ABB RAPID module: 8947b821.mod

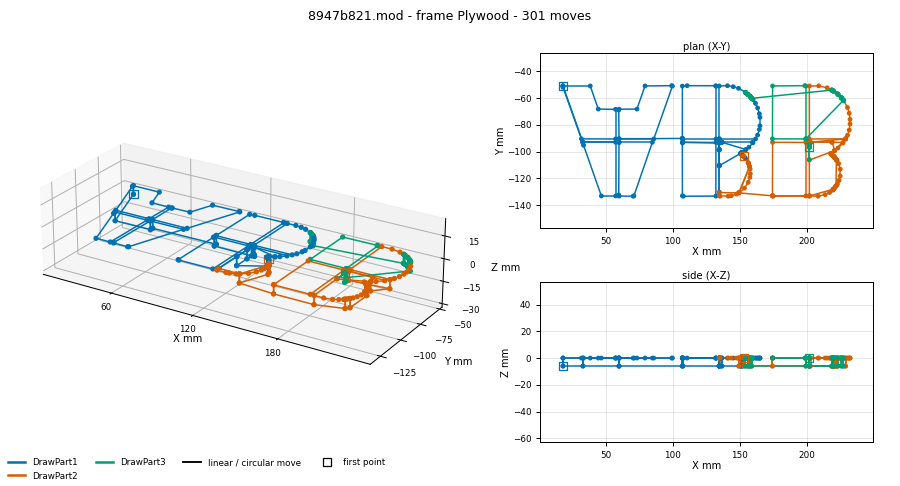
[picture p0: tool path of 8947b821.mod in frame Plywood, 301 of 303 moves have a stored position in this frame; points joined in program order, loops and branches not executed]
MODULE ImageDraw
  ! Generated 2026-10-07 09:33 for ABB GoFa CRB 15000-5/0.95: 40 strokes
  ! Page 250 x 180 mm. Work object Plywood: Z points DOWN, so pen-up is -Z and the tool uses orientation [1,0,0,0].
  ! Uses the tool 'tcp' and work object 'Plywood' that already exist on the controller.
  CONST robtarget pOrigin:=[[0,0,0],[1,0,0,0],[0,0,0,0],[9E9,9E9,9E9,9E9,9E9,9E9]];
  CONST jointtarget jHome:=[[0,0,0,0,30,0],[9E9,9E9,9E9,9E9,9E9,9E9]];
  CONST speeddata vTravel:=[250,200,5000,1000];

  PROC main()
    SingArea\Wrist;
    ConfL\Off;
    ConfJ\Off;
    MoveAbsJ jHome\NoEOffs,vTravel,fine,tcp;
    DrawPart1;
    DrawPart2;
    DrawPart3;
    MoveAbsJ jHome\NoEOffs,vTravel,fine,tcp;
  ENDPROC

  PROC DrawPart1()
    MoveL Offs(pOrigin,17.75,-50.83,-6.00),vTravel,z5,tcp\WObj:=Plywood;
    MoveL Offs(pOrigin,17.75,-50.83,-0.00),v60,z0,tcp\WObj:=Plywood;
    MoveL Offs(pOrigin,38.15,-50.83,-0.00),v40,z0,tcp\WObj:=Plywood;
    MoveL Offs(pOrigin,44.15,-68.12,-0.00),v40,z0,tcp\WObj:=Plywood;
    MoveL Offs(pOrigin,57.05,-68.32,-0.00),v40,z0,tcp\WObj:=Plywood;
    MoveL Offs(pOrigin,57.05,-90.47,-0.00),v40,z0,tcp\WObj:=Plywood;
    MoveL Offs(pOrigin,31.55,-90.38,-0.00),v40,z0,tcp\WObj:=Plywood;
    MoveL Offs(pOrigin,17.80,-51.83,-0.00),v40,z0,tcp\WObj:=Plywood;
    MoveL Offs(pOrigin,17.75,-50.83,-0.00),v40,fine,tcp\WObj:=Plywood;
    MoveL Offs(pOrigin,17.75,-50.83,-6.00),v60,z5,tcp\WObj:=Plywood;
    MoveL Offs(pOrigin,32.65,-92.97,-6.00),vTravel,z5,tcp\WObj:=Plywood;
    MoveL Offs(pOrigin,32.65,-92.97,-0.00),v60,z0,tcp\WObj:=Plywood;
    MoveL Offs(pOrigin,33.15,-95.18,-0.00),v40,z0,tcp\WObj:=Plywood;
    MoveL Offs(pOrigin,46.45,-133.07,-0.00),v40,z0,tcp\WObj:=Plywood;
    MoveL Offs(pOrigin,57.15,-133.07,-0.00),v40,z0,tcp\WObj:=Plywood;
    MoveL Offs(pOrigin,57.15,-92.97,-0.00),v40,z0,tcp\WObj:=Plywood;
    MoveL Offs(pOrigin,32.65,-92.97,-0.00),v40,fine,tcp\WObj:=Plywood;
    MoveL Offs(pOrigin,32.65,-92.97,-6.00),v60,z5,tcp\WObj:=Plywood;
    MoveL Offs(pOrigin,59.65,-92.97,-6.00),vTravel,z5,tcp\WObj:=Plywood;
    MoveL Offs(pOrigin,59.65,-92.97,-0.00),v60,z0,tcp\WObj:=Plywood;
    MoveL Offs(pOrigin,59.45,-132.38,-0.00),v40,z0,tcp\WObj:=Plywood;
    MoveL Offs(pOrigin,59.75,-133.18,-0.00),v40,z0,tcp\WObj:=Plywood;
    MoveL Offs(pOrigin,70.25,-133.27,-0.00),v40,z0,tcp\WObj:=Plywood;
    MoveL Offs(pOrigin,70.80,-132.98,-0.00),v40,z0,tcp\WObj:=Plywood;
    MoveL Offs(pOrigin,84.60,-92.97,-0.00),v40,z0,tcp\WObj:=Plywood;
    MoveL Offs(pOrigin,59.65,-92.97,-0.00),v40,fine,tcp\WObj:=Plywood;
    MoveL Offs(pOrigin,59.65,-92.97,-6.00),v60,z5,tcp\WObj:=Plywood;
    MoveL Offs(pOrigin,59.65,-90.38,-6.00),vTravel,z5,tcp\WObj:=Plywood;
    MoveL Offs(pOrigin,59.65,-90.38,-0.00),v60,z0,tcp\WObj:=Plywood;
    MoveL Offs(pOrigin,59.45,-68.78,-0.00),v40,z0,tcp\WObj:=Plywood;
    MoveL Offs(pOrigin,59.75,-68.22,-0.00),v40,z0,tcp\WObj:=Plywood;
    MoveL Offs(pOrigin,73.05,-68.12,-0.00),v40,z0,tcp\WObj:=Plywood;
    MoveL Offs(pOrigin,79.10,-50.83,-0.00),v40,z0,tcp\WObj:=Plywood;
    MoveL Offs(pOrigin,99.05,-50.62,-0.00),v40,z0,tcp\WObj:=Plywood;
    MoveL Offs(pOrigin,99.60,-50.92,-0.00),v40,z0,tcp\WObj:=Plywood;
    MoveL Offs(pOrigin,85.65,-90.47,-0.00),v40,z0,tcp\WObj:=Plywood;
    MoveL Offs(pOrigin,59.65,-90.38,-0.00),v40,fine,tcp\WObj:=Plywood;
    MoveL Offs(pOrigin,59.65,-90.38,-6.00),v60,z5,tcp\WObj:=Plywood;
    MoveL Offs(pOrigin,107.00,-90.07,-6.00),vTravel,z5,tcp\WObj:=Plywood;
    MoveL Offs(pOrigin,107.00,-90.07,-0.00),v60,z0,tcp\WObj:=Plywood;
    MoveL Offs(pOrigin,107.05,-50.92,-0.00),v40,z0,tcp\WObj:=Plywood;
    MoveL Offs(pOrigin,110.60,-50.62,-0.00),v40,z0,tcp\WObj:=Plywood;
    MoveL Offs(pOrigin,131.90,-50.67,-0.00),v40,z0,tcp\WObj:=Plywood;
    MoveL Offs(pOrigin,132.20,-51.08,-0.00),v40,z0,tcp\WObj:=Plywood;
    MoveL Offs(pOrigin,132.15,-90.47,-0.00),v40,z0,tcp\WObj:=Plywood;
    MoveL Offs(pOrigin,107.30,-90.47,-0.00),v40,z0,tcp\WObj:=Plywood;
    MoveL Offs(pOrigin,107.00,-90.07,-0.00),v40,fine,tcp\WObj:=Plywood;
    MoveL Offs(pOrigin,107.00,-90.07,-6.00),v60,z5,tcp\WObj:=Plywood;
    MoveL Offs(pOrigin,107.30,-92.97,-6.00),vTravel,z5,tcp\WObj:=Plywood;
    MoveL Offs(pOrigin,107.30,-92.97,-0.00),v60,z0,tcp\WObj:=Plywood;
    MoveL Offs(pOrigin,132.15,-93.07,-0.00),v40,z0,tcp\WObj:=Plywood;
    MoveL Offs(pOrigin,132.05,-133.18,-0.00),v40,z0,tcp\WObj:=Plywood;
    MoveL Offs(pOrigin,107.75,-133.27,-0.00),v40,z0,tcp\WObj:=Plywood;
    MoveL Offs(pOrigin,107.05,-132.98,-0.00),v40,z0,tcp\WObj:=Plywood;
    MoveL Offs(pOrigin,107.00,-93.38,-0.00),v40,z0,tcp\WObj:=Plywood;
    MoveL Offs(pOrigin,107.30,-92.97,-0.00),v40,fine,tcp\WObj:=Plywood;
    MoveL Offs(pOrigin,107.30,-92.97,-6.00),v60,z5,tcp\WObj:=Plywood;
    MoveL Offs(pOrigin,134.60,-93.53,-6.00),vTravel,z5,tcp\WObj:=Plywood;
    MoveL Offs(pOrigin,134.60,-93.53,-0.00),v60,z0,tcp\WObj:=Plywood;
    MoveL Offs(pOrigin,134.60,-98.18,-0.00),v40,z0,tcp\WObj:=Plywood;
    MoveL Offs(pOrigin,134.60,-93.53,-0.00),v40,z0,tcp\WObj:=Plywood;
    MoveL Offs(pOrigin,135.05,-92.93,-0.00),v40,z0,tcp\WObj:=Plywood;
    MoveL Offs(pOrigin,136.25,-92.93,-0.00),v40,z0,tcp\WObj:=Plywood;
    MoveL Offs(pOrigin,135.05,-92.93,-0.00),v40,fine,tcp\WObj:=Plywood;
    MoveL Offs(pOrigin,135.05,-92.93,-6.00),v60,z5,tcp\WObj:=Plywood;
    MoveL Offs(pOrigin,136.55,-92.93,-6.00),vTravel,z5,tcp\WObj:=Plywood;
    MoveL Offs(pOrigin,136.55,-92.93,-0.00),v60,z0,tcp\WObj:=Plywood;
    MoveL Offs(pOrigin,159.50,-92.93,-0.00),v40,z0,tcp\WObj:=Plywood;
    MoveL Offs(pOrigin,159.80,-93.38,-0.00),v40,z0,tcp\WObj:=Plywood;
    MoveL Offs(pOrigin,156.80,-96.62,-0.00),v40,z0,tcp\WObj:=Plywood;
    MoveL Offs(pOrigin,154.60,-98.38,-0.00),v40,z0,tcp\WObj:=Plywood;
    MoveL Offs(pOrigin,136.55,-92.93,-0.00),v40,fine,tcp\WObj:=Plywood;
    MoveL Offs(pOrigin,136.55,-92.93,-6.00),v60,z5,tcp\WObj:=Plywood;
    MoveL Offs(pOrigin,134.65,-90.47,-6.00),vTravel,z5,tcp\WObj:=Plywood;
    MoveL Offs(pOrigin,134.65,-90.47,-0.00),v60,z0,tcp\WObj:=Plywood;
    MoveL Offs(pOrigin,161.75,-90.47,-0.00),v40,z0,tcp\WObj:=Plywood;
    MoveL Offs(pOrigin,163.30,-87.53,-0.00),v40,z0,tcp\WObj:=Plywood;
    MoveL Offs(pOrigin,164.60,-83.32,-0.00),v40,z0,tcp\WObj:=Plywood;
    MoveL Offs(pOrigin,165.05,-80.62,-0.00),v40,z0,tcp\WObj:=Plywood;
    MoveL Offs(pOrigin,165.05,-74.32,-0.00),v40,z0,tcp\WObj:=Plywood;
    MoveL Offs(pOrigin,164.60,-71.62,-0.00),v40,z0,tcp\WObj:=Plywood;
    MoveL Offs(pOrigin,163.30,-67.28,-0.00),v40,z0,tcp\WObj:=Plywood;
    MoveL Offs(pOrigin,161.70,-63.83,-0.00),v40,z0,tcp\WObj:=Plywood;
    MoveL Offs(pOrigin,159.95,-61.12,-0.00),v40,z0,tcp\WObj:=Plywood;
    MoveL Offs(pOrigin,157.55,-58.28,-0.00),v40,z0,tcp\WObj:=Plywood;
    MoveL Offs(pOrigin,154.55,-55.72,-0.00),v40,z0,tcp\WObj:=Plywood;
    MoveL Offs(pOrigin,149.00,-52.62,-0.00),v40,z0,tcp\WObj:=Plywood;
    MoveL Offs(pOrigin,145.10,-51.38,-0.00),v40,z0,tcp\WObj:=Plywood;
    MoveL Offs(pOrigin,140.75,-50.62,-0.00),v40,z0,tcp\WObj:=Plywood;
    MoveL Offs(pOrigin,134.65,-50.83,-0.00),v40,z0,tcp\WObj:=Plywood;
    MoveL Offs(pOrigin,134.65,-90.47,-0.00),v40,fine,tcp\WObj:=Plywood;
    MoveL Offs(pOrigin,134.65,-90.47,-6.00),v60,z5,tcp\WObj:=Plywood;
    MoveL Offs(pOrigin,134.60,-98.62,-6.00),vTravel,z5,tcp\WObj:=Plywood;
    MoveL Offs(pOrigin,134.60,-98.62,-0.00),v60,z0,tcp\WObj:=Plywood;
    MoveL Offs(pOrigin,134.60,-110.03,-0.00),v40,z0,tcp\WObj:=Plywood;
    MoveL Offs(pOrigin,134.60,-98.62,-0.00),v40,fine,tcp\WObj:=Plywood;
    MoveL Offs(pOrigin,134.60,-98.62,-6.00),v60,z5,tcp\WObj:=Plywood;
    MoveL Offs(pOrigin,134.60,-110.47,-6.00),vTravel,z5,tcp\WObj:=Plywood;
    MoveL Offs(pOrigin,134.60,-110.47,-0.00),v60,z0,tcp\WObj:=Plywood;
    MoveL Offs(pOrigin,134.60,-130.12,-0.00),v40,z0,tcp\WObj:=Plywood;
    MoveL Offs(pOrigin,134.60,-110.47,-0.00),v40,fine,tcp\WObj:=Plywood;
    MoveL Offs(pOrigin,134.60,-110.47,-6.00),v60,z5,tcp\WObj:=Plywood;
    MoveL Offs(pOrigin,150.50,-101.32,-6.00),vTravel,z5,tcp\WObj:=Plywood;
    MoveL Offs(pOrigin,150.50,-101.32,-0.00),v60,z0,tcp\WObj:=Plywood;
    MoveL Offs(pOrigin,151.10,-100.68,-0.00),v40,z0,tcp\WObj:=Plywood;
    MoveL Offs(pOrigin,151.80,-102.57,-0.00),v40,z0,tcp\WObj:=Plywood;
    MoveL Offs(pOrigin,150.50,-101.32,-0.00),v40,fine,tcp\WObj:=Plywood;
    MoveL Offs(pOrigin,150.50,-101.32,-6.00),v60,z5,tcp\WObj:=Plywood;
    MoveL Offs(pOrigin,151.45,-100.47,-6.00),vTravel,z5,tcp\WObj:=Plywood;
    MoveL Offs(pOrigin,151.45,-100.47,-0.00),v60,z0,tcp\WObj:=Plywood;
    MoveL Offs(pOrigin,154.30,-98.53,-0.00),v40,z0,tcp\WObj:=Plywood;
    MoveL Offs(pOrigin,151.45,-100.47,-0.00),v40,fine,tcp\WObj:=Plywood;
    MoveL Offs(pOrigin,151.45,-100.47,-6.00),v60,z5,tcp\WObj:=Plywood;
    MoveL Offs(pOrigin,152.05,-102.78,-6.00),vTravel,z5,tcp\WObj:=Plywood;
    MoveL Offs(pOrigin,152.05,-102.78,-0.00),v60,z0,tcp\WObj:=Plywood;
    MoveL Offs(pOrigin,154.25,-105.07,-0.00),v40,z0,tcp\WObj:=Plywood;
    MoveL Offs(pOrigin,156.25,-108.18,-0.00),v40,z0,tcp\WObj:=Plywood;
    MoveL Offs(pOrigin,152.05,-102.78,-0.00),v40,z0,tcp\WObj:=Plywood;
    MoveL Offs(pOrigin,152.90,-103.43,-0.00),v40,z0,tcp\WObj:=Plywood;
    MoveL Offs(pOrigin,153.50,-104.03,-0.00),v40,z0,tcp\WObj:=Plywood;
  ENDPROC

  PROC DrawPart2()
    MoveL Offs(pOrigin,152.90,-103.43,-0.00),v40,fine,tcp\WObj:=Plywood;
    MoveL Offs(pOrigin,152.90,-103.43,-6.00),v60,z5,tcp\WObj:=Plywood;
    MoveL Offs(pOrigin,156.35,-108.53,-6.00),vTravel,z5,tcp\WObj:=Plywood;
    MoveL Offs(pOrigin,156.35,-108.53,-0.00),v60,z0,tcp\WObj:=Plywood;
    MoveL Offs(pOrigin,157.20,-110.78,-0.00),v40,z0,tcp\WObj:=Plywood;
    MoveL Offs(pOrigin,156.35,-108.53,-0.00),v40,fine,tcp\WObj:=Plywood;
    MoveL Offs(pOrigin,156.35,-108.53,-6.00),v60,z5,tcp\WObj:=Plywood;
    MoveL Offs(pOrigin,157.25,-111.22,-6.00),vTravel,z5,tcp\WObj:=Plywood;
    MoveL Offs(pOrigin,157.25,-111.22,-0.00),v60,z0,tcp\WObj:=Plywood;
    MoveL Offs(pOrigin,157.70,-113.03,-0.00),v40,z0,tcp\WObj:=Plywood;
    MoveL Offs(pOrigin,157.85,-116.47,-0.00),v40,z0,tcp\WObj:=Plywood;
    MoveL Offs(pOrigin,157.55,-119.18,-0.00),v40,z0,tcp\WObj:=Plywood;
    MoveL Offs(pOrigin,156.30,-122.93,-0.00),v40,z0,tcp\WObj:=Plywood;
    MoveL Offs(pOrigin,153.45,-127.28,-0.00),v40,z0,tcp\WObj:=Plywood;
    MoveL Offs(pOrigin,149.50,-130.62,-0.00),v40,z0,tcp\WObj:=Plywood;
    MoveL Offs(pOrigin,157.25,-111.22,-0.00),v40,fine,tcp\WObj:=Plywood;
    MoveL Offs(pOrigin,157.25,-111.22,-6.00),v60,z5,tcp\WObj:=Plywood;
    MoveL Offs(pOrigin,149.20,-130.77,-6.00),vTravel,z5,tcp\WObj:=Plywood;
    MoveL Offs(pOrigin,149.20,-130.77,-0.00),v60,z0,tcp\WObj:=Plywood;
    MoveL Offs(pOrigin,134.60,-130.57,-0.00),v40,z0,tcp\WObj:=Plywood;
    MoveL Offs(pOrigin,134.60,-132.98,-0.00),v40,z0,tcp\WObj:=Plywood;
    MoveL Offs(pOrigin,135.20,-133.27,-0.00),v40,z0,tcp\WObj:=Plywood;
    MoveL Offs(pOrigin,141.35,-133.27,-0.00),v40,z0,tcp\WObj:=Plywood;
    MoveL Offs(pOrigin,143.60,-132.98,-0.00),v40,z0,tcp\WObj:=Plywood;
    MoveL Offs(pOrigin,147.50,-131.73,-0.00),v40,z0,tcp\WObj:=Plywood;
    MoveL Offs(pOrigin,149.20,-130.77,-0.00),v40,fine,tcp\WObj:=Plywood;
    MoveL Offs(pOrigin,149.20,-130.77,-6.00),v60,z5,tcp\WObj:=Plywood;
    MoveL Offs(pOrigin,174.40,-132.98,-6.00),vTravel,z5,tcp\WObj:=Plywood;
    MoveL Offs(pOrigin,174.40,-132.98,-0.00),v60,z0,tcp\WObj:=Plywood;
    MoveL Offs(pOrigin,174.50,-92.97,-0.00),v40,z0,tcp\WObj:=Plywood;
    MoveL Offs(pOrigin,199.35,-93.07,-0.00),v40,z0,tcp\WObj:=Plywood;
    MoveL Offs(pOrigin,199.35,-133.07,-0.00),v40,z0,tcp\WObj:=Plywood;
    MoveL Offs(pOrigin,174.95,-133.27,-0.00),v40,z0,tcp\WObj:=Plywood;
    MoveL Offs(pOrigin,174.40,-132.98,-0.00),v40,fine,tcp\WObj:=Plywood;
    MoveL Offs(pOrigin,174.40,-132.98,-6.00),v60,z5,tcp\WObj:=Plywood;
    MoveL Offs(pOrigin,202.00,-133.07,-6.00),vTravel,z5,tcp\WObj:=Plywood;
    MoveL Offs(pOrigin,202.00,-133.07,-0.00),v60,z0,tcp\WObj:=Plywood;
    MoveL Offs(pOrigin,208.55,-133.27,-0.00),v40,z0,tcp\WObj:=Plywood;
    MoveL Offs(pOrigin,213.80,-132.12,-0.00),v40,z0,tcp\WObj:=Plywood;
    MoveL Offs(pOrigin,217.10,-130.48,-0.00),v40,z0,tcp\WObj:=Plywood;
    MoveL Offs(pOrigin,219.35,-128.77,-0.00),v40,z0,tcp\WObj:=Plywood;
    MoveL Offs(pOrigin,220.70,-127.43,-0.00),v40,z0,tcp\WObj:=Plywood;
    MoveL Offs(pOrigin,223.00,-124.12,-0.00),v40,z0,tcp\WObj:=Plywood;
    MoveL Offs(pOrigin,224.20,-121.43,-0.00),v40,z0,tcp\WObj:=Plywood;
    MoveL Offs(pOrigin,225.05,-118.12,-0.00),v40,z0,tcp\WObj:=Plywood;
    MoveL Offs(pOrigin,225.05,-113.03,-0.00),v40,z0,tcp\WObj:=Plywood;
    MoveL Offs(pOrigin,223.90,-108.97,-0.00),v40,z0,tcp\WObj:=Plywood;
    MoveL Offs(pOrigin,222.70,-106.57,-0.00),v40,z0,tcp\WObj:=Plywood;
    MoveL Offs(pOrigin,220.55,-103.72,-0.00),v40,z0,tcp\WObj:=Plywood;
    MoveL Offs(pOrigin,217.75,-101.32,-0.00),v40,z0,tcp\WObj:=Plywood;
    MoveL Offs(pOrigin,220.60,-99.28,-0.00),v40,z0,tcp\WObj:=Plywood;
    MoveL Offs(pOrigin,201.95,-106.28,-0.00),v40,z0,tcp\WObj:=Plywood;
    MoveL Offs(pOrigin,202.00,-133.07,-0.00),v40,fine,tcp\WObj:=Plywood;
    MoveL Offs(pOrigin,202.00,-133.07,-6.00),v60,z5,tcp\WObj:=Plywood;
    MoveL Offs(pOrigin,219.95,-128.02,-6.00),vTravel,z5,tcp\WObj:=Plywood;
    MoveL Offs(pOrigin,219.95,-128.02,-0.00),v60,z0,tcp\WObj:=Plywood;
    MoveL Offs(pOrigin,219.50,-128.48,-0.00),v40,z0,tcp\WObj:=Plywood;
    MoveL Offs(pOrigin,219.95,-128.02,-0.00),v40,fine,tcp\WObj:=Plywood;
    MoveL Offs(pOrigin,219.95,-128.02,-6.00),v60,z5,tcp\WObj:=Plywood;
    MoveL Offs(pOrigin,221.90,-125.62,-6.00),vTravel,z5,tcp\WObj:=Plywood;
    MoveL Offs(pOrigin,221.90,-125.62,-0.00),v60,z0,tcp\WObj:=Plywood;
    MoveL Offs(pOrigin,221.30,-126.38,-0.00),v40,z0,tcp\WObj:=Plywood;
    MoveL Offs(pOrigin,221.90,-125.62,-0.00),v40,fine,tcp\WObj:=Plywood;
    MoveL Offs(pOrigin,221.90,-125.62,-6.00),v60,z5,tcp\WObj:=Plywood;
    MoveL Offs(pOrigin,222.20,-105.97,-6.00),vTravel,z5,tcp\WObj:=Plywood;
    MoveL Offs(pOrigin,222.20,-105.97,-0.00),v60,z0,tcp\WObj:=Plywood;
    MoveL Offs(pOrigin,222.50,-106.43,-0.00),v40,z0,tcp\WObj:=Plywood;
    MoveL Offs(pOrigin,222.20,-105.97,-0.00),v40,fine,tcp\WObj:=Plywood;
    MoveL Offs(pOrigin,222.20,-105.97,-6.00),v60,z5,tcp\WObj:=Plywood;
    MoveL Offs(pOrigin,220.85,-104.32,-6.00),vTravel,z5,tcp\WObj:=Plywood;
    MoveL Offs(pOrigin,220.85,-104.32,-0.00),v60,z0,tcp\WObj:=Plywood;
    MoveL Offs(pOrigin,221.45,-104.93,-0.00),v40,z0,tcp\WObj:=Plywood;
    MoveL Offs(pOrigin,220.85,-104.32,-0.00),v40,fine,tcp\WObj:=Plywood;
    MoveL Offs(pOrigin,220.85,-104.32,-6.00),v60,z5,tcp\WObj:=Plywood;
    MoveL Offs(pOrigin,219.80,-103.12,-6.00),vTravel,z5,tcp\WObj:=Plywood;
    MoveL Offs(pOrigin,219.80,-103.12,-0.00),v60,z0,tcp\WObj:=Plywood;
    MoveL Offs(pOrigin,220.55,-103.88,-0.00),v40,z0,tcp\WObj:=Plywood;
    MoveL Offs(pOrigin,219.80,-103.12,-0.00),v40,fine,tcp\WObj:=Plywood;
    MoveL Offs(pOrigin,219.80,-103.12,-6.00),v60,z5,tcp\WObj:=Plywood;
    MoveL Offs(pOrigin,218.60,-102.07,-6.00),vTravel,z5,tcp\WObj:=Plywood;
    MoveL Offs(pOrigin,218.60,-102.07,-0.00),v60,z0,tcp\WObj:=Plywood;
    MoveL Offs(pOrigin,219.50,-102.97,-0.00),v40,z0,tcp\WObj:=Plywood;
    MoveL Offs(pOrigin,218.60,-102.07,-0.00),v40,fine,tcp\WObj:=Plywood;
    MoveL Offs(pOrigin,218.60,-102.07,-6.00),v60,z5,tcp\WObj:=Plywood;
    MoveL Offs(pOrigin,220.90,-99.12,-6.00),vTravel,z5,tcp\WObj:=Plywood;
    MoveL Offs(pOrigin,220.90,-99.12,-0.00),v60,z0,tcp\WObj:=Plywood;
    MoveL Offs(pOrigin,219.05,-92.93,-0.00),v40,z0,tcp\WObj:=Plywood;
    MoveL Offs(pOrigin,227.10,-93.07,-0.00),v40,z0,tcp\WObj:=Plywood;
    MoveL Offs(pOrigin,227.10,-93.53,-0.00),v40,z0,tcp\WObj:=Plywood;
    MoveL Offs(pOrigin,223.40,-97.22,-0.00),v40,z0,tcp\WObj:=Plywood;
    MoveL Offs(pOrigin,220.90,-99.12,-0.00),v40,fine,tcp\WObj:=Plywood;
    MoveL Offs(pOrigin,220.90,-99.12,-6.00),v60,z5,tcp\WObj:=Plywood;
    MoveL Offs(pOrigin,229.10,-90.38,-6.00),vTravel,z5,tcp\WObj:=Plywood;
    MoveL Offs(pOrigin,229.10,-90.38,-0.00),v60,z0,tcp\WObj:=Plywood;
    MoveL Offs(pOrigin,230.55,-87.68,-0.00),v40,z0,tcp\WObj:=Plywood;
    MoveL Offs(pOrigin,231.80,-83.78,-0.00),v40,z0,tcp\WObj:=Plywood;
    MoveL Offs(pOrigin,232.40,-79.28,-0.00),v40,z0,tcp\WObj:=Plywood;
    MoveL Offs(pOrigin,232.40,-75.82,-0.00),v40,z0,tcp\WObj:=Plywood;
    MoveL Offs(pOrigin,231.80,-71.18,-0.00),v40,z0,tcp\WObj:=Plywood;
    MoveL Offs(pOrigin,230.50,-66.97,-0.00),v40,z0,tcp\WObj:=Plywood;
    MoveL Offs(pOrigin,227.45,-61.42,-0.00),v40,z0,tcp\WObj:=Plywood;
    MoveL Offs(pOrigin,225.80,-59.33,-0.00),v40,z0,tcp\WObj:=Plywood;
    MoveL Offs(pOrigin,222.65,-56.33,-0.00),v40,z0,tcp\WObj:=Plywood;
    MoveL Offs(pOrigin,218.90,-53.88,-0.00),v40,z0,tcp\WObj:=Plywood;
    MoveL Offs(pOrigin,215.30,-52.22,-0.00),v40,z0,tcp\WObj:=Plywood;
    MoveL Offs(pOrigin,209.00,-50.78,-0.00),v40,z0,tcp\WObj:=Plywood;
    MoveL Offs(pOrigin,201.95,-50.83,-0.00),v40,z0,tcp\WObj:=Plywood;
    MoveL Offs(pOrigin,202.00,-90.47,-0.00),v40,z0,tcp\WObj:=Plywood;
    MoveL Offs(pOrigin,229.10,-90.38,-0.00),v40,fine,tcp\WObj:=Plywood;
    MoveL Offs(pOrigin,229.10,-90.38,-6.00),v60,z5,tcp\WObj:=Plywood;
    MoveL Offs(pOrigin,202.85,-92.93,-6.00),vTravel,z5,tcp\WObj:=Plywood;
    MoveL Offs(pOrigin,202.85,-92.93,-0.00),v60,z0,tcp\WObj:=Plywood;
    MoveL Offs(pOrigin,218.60,-92.93,-0.00),v40,z0,tcp\WObj:=Plywood;
    MoveL Offs(pOrigin,202.85,-92.93,-0.00),v40,z0,tcp\WObj:=Plywood;
    MoveL Offs(pOrigin,201.95,-93.53,-0.00),v40,z0,tcp\WObj:=Plywood;
    MoveL Offs(pOrigin,201.95,-94.72,-0.00),v40,z0,tcp\WObj:=Plywood;
    MoveL Offs(pOrigin,201.95,-93.53,-0.00),v40,fine,tcp\WObj:=Plywood;
    MoveL Offs(pOrigin,201.95,-93.53,-6.00),v60,z5,tcp\WObj:=Plywood;
    MoveL Offs(pOrigin,201.95,-94.88,-6.00),vTravel,z5,tcp\WObj:=Plywood;
    MoveL Offs(pOrigin,201.95,-94.88,-0.00),v60,z0,tcp\WObj:=Plywood;
  ENDPROC

  PROC DrawPart3()
    MoveL Offs(pOrigin,201.95,-96.38,-0.00),v40,z0,tcp\WObj:=Plywood;
    MoveL Offs(pOrigin,201.95,-94.88,-0.00),v40,fine,tcp\WObj:=Plywood;
    MoveL Offs(pOrigin,201.95,-94.88,-6.00),v60,z5,tcp\WObj:=Plywood;
    MoveL Offs(pOrigin,201.95,-96.68,-6.00),vTravel,z5,tcp\WObj:=Plywood;
    MoveL Offs(pOrigin,201.95,-96.68,-0.00),v60,z0,tcp\WObj:=Plywood;
    MoveL Offs(pOrigin,201.95,-105.82,-0.00),v40,z0,tcp\WObj:=Plywood;
    MoveL Offs(pOrigin,201.95,-96.68,-0.00),v40,fine,tcp\WObj:=Plywood;
    MoveL Offs(pOrigin,201.95,-96.68,-6.00),v60,z5,tcp\WObj:=Plywood;
    MoveL Offs(pOrigin,199.35,-90.47,-6.00),vTravel,z5,tcp\WObj:=Plywood;
    MoveL Offs(pOrigin,199.35,-90.47,-0.00),v60,z0,tcp\WObj:=Plywood;
    MoveL Offs(pOrigin,174.40,-90.38,-0.00),v40,z0,tcp\WObj:=Plywood;
    MoveL Offs(pOrigin,174.50,-50.83,-0.00),v40,z0,tcp\WObj:=Plywood;
    MoveL Offs(pOrigin,198.65,-50.62,-0.00),v40,z0,tcp\WObj:=Plywood;
    MoveL Offs(pOrigin,199.35,-50.92,-0.00),v40,z0,tcp\WObj:=Plywood;
    MoveL Offs(pOrigin,199.35,-90.47,-0.00),v40,fine,tcp\WObj:=Plywood;
    MoveL Offs(pOrigin,199.35,-90.47,-6.00),v60,z5,tcp\WObj:=Plywood;
    MoveL Offs(pOrigin,227.45,-61.58,-6.00),vTravel,z5,tcp\WObj:=Plywood;
    MoveL Offs(pOrigin,227.45,-61.58,-0.00),v60,z0,tcp\WObj:=Plywood;
    MoveL Offs(pOrigin,227.75,-62.03,-0.00),v40,z0,tcp\WObj:=Plywood;
    MoveL Offs(pOrigin,227.45,-61.58,-0.00),v40,fine,tcp\WObj:=Plywood;
    MoveL Offs(pOrigin,227.45,-61.58,-6.00),v60,z5,tcp\WObj:=Plywood;
    MoveL Offs(pOrigin,225.95,-59.78,-6.00),vTravel,z5,tcp\WObj:=Plywood;
    MoveL Offs(pOrigin,225.95,-59.78,-0.00),v60,z0,tcp\WObj:=Plywood;
    MoveL Offs(pOrigin,226.70,-60.53,-0.00),v40,z0,tcp\WObj:=Plywood;
    MoveL Offs(pOrigin,225.95,-59.78,-0.00),v40,fine,tcp\WObj:=Plywood;
    MoveL Offs(pOrigin,225.95,-59.78,-6.00),v60,z5,tcp\WObj:=Plywood;
    MoveL Offs(pOrigin,223.40,-57.12,-6.00),vTravel,z5,tcp\WObj:=Plywood;
    MoveL Offs(pOrigin,223.40,-57.12,-0.00),v60,z0,tcp\WObj:=Plywood;
    MoveL Offs(pOrigin,225.65,-59.33,-0.00),v40,z0,tcp\WObj:=Plywood;
    MoveL Offs(pOrigin,223.40,-57.12,-0.00),v40,fine,tcp\WObj:=Plywood;
    MoveL Offs(pOrigin,223.40,-57.12,-6.00),v60,z5,tcp\WObj:=Plywood;
    MoveL Offs(pOrigin,219.80,-54.53,-6.00),vTravel,z5,tcp\WObj:=Plywood;
    MoveL Offs(pOrigin,219.80,-54.53,-0.00),v60,z0,tcp\WObj:=Plywood;
    MoveL Offs(pOrigin,220.25,-54.83,-0.00),v40,z0,tcp\WObj:=Plywood;
    MoveL Offs(pOrigin,219.80,-54.53,-0.00),v40,fine,tcp\WObj:=Plywood;
    MoveL Offs(pOrigin,219.80,-54.53,-6.00),v60,z5,tcp\WObj:=Plywood;
    MoveL Offs(pOrigin,218.75,-53.92,-6.00),vTravel,z5,tcp\WObj:=Plywood;
    MoveL Offs(pOrigin,218.75,-53.92,-0.00),v60,z0,tcp\WObj:=Plywood;
    MoveL Offs(pOrigin,219.20,-54.22,-0.00),v40,z0,tcp\WObj:=Plywood;
    MoveL Offs(pOrigin,218.75,-53.92,-0.00),v40,fine,tcp\WObj:=Plywood;
    MoveL Offs(pOrigin,218.75,-53.92,-6.00),v60,z5,tcp\WObj:=Plywood;
    MoveL Offs(pOrigin,158.90,-60.08,-6.00),vTravel,z5,tcp\WObj:=Plywood;
    MoveL Offs(pOrigin,158.90,-60.08,-0.00),v60,z0,tcp\WObj:=Plywood;
    MoveL Offs(pOrigin,159.35,-60.53,-0.00),v40,z0,tcp\WObj:=Plywood;
    MoveL Offs(pOrigin,158.90,-60.08,-0.00),v40,fine,tcp\WObj:=Plywood;
    MoveL Offs(pOrigin,158.90,-60.08,-6.00),v60,z5,tcp\WObj:=Plywood;
    MoveL Offs(pOrigin,157.85,-58.88,-6.00),vTravel,z5,tcp\WObj:=Plywood;
    MoveL Offs(pOrigin,157.85,-58.88,-0.00),v60,z0,tcp\WObj:=Plywood;
    MoveL Offs(pOrigin,158.75,-59.78,-0.00),v40,z0,tcp\WObj:=Plywood;
    MoveL Offs(pOrigin,157.85,-58.88,-0.00),v40,fine,tcp\WObj:=Plywood;
    MoveL Offs(pOrigin,157.85,-58.88,-6.00),v60,z5,tcp\WObj:=Plywood;
    MoveL Offs(pOrigin,155.90,-57.08,-6.00),vTravel,z5,tcp\WObj:=Plywood;
    MoveL Offs(pOrigin,155.90,-57.08,-0.00),v60,z0,tcp\WObj:=Plywood;
    MoveL Offs(pOrigin,156.95,-57.97,-0.00),v40,z0,tcp\WObj:=Plywood;
    MoveL Offs(pOrigin,155.90,-57.08,-0.00),v40,fine,tcp\WObj:=Plywood;
    MoveL Offs(pOrigin,155.90,-57.08,-6.00),v60,z5,tcp\WObj:=Plywood;
    MoveL Offs(pOrigin,154.10,-55.58,-6.00),vTravel,z5,tcp\WObj:=Plywood;
    MoveL Offs(pOrigin,154.10,-55.58,-0.00),v60,z0,tcp\WObj:=Plywood;
    MoveL Offs(pOrigin,154.85,-56.17,-0.00),v40,z0,tcp\WObj:=Plywood;
    MoveL Offs(pOrigin,154.10,-55.58,-0.00),v40,fine,tcp\WObj:=Plywood;
    MoveL Offs(pOrigin,154.10,-55.58,-6.00),v60,z5,tcp\WObj:=Plywood;
  ENDPROC

ENDMODULE
